FUNCTION_BLOCK FB_AdjustablePump IMPLEMENTS I_AdjustablePump

VAR
	bRunning : BOOL;
	fTotalVolume : REAL;
	fFlowRate : REAL := 20;
END_VAR

IF bRunning THEN
	fTotalVolume := fTotalVolume + fFlowRate;
END_IF

{warning 'add method implementation '}
METHOD GetFlowRate : REAL
GetFlowRate := fFlowRate;
END_METHOD

{warning 'add method implementation '}
METHOD GetTotalVolume : REAL
GetTotalVolume := fTotalVolume;
END_METHOD

METHOD SetFlowRate : BOOL
VAR_INPUT
	fNewRate : REAL;
END_VAR
fFlowRate := fNewRate;
END_METHOD

{warning 'add method implementation '}
METHOD Start : BOOL
Start := bRunning := TRUE;
END_METHOD

{warning 'add method implementation '}
METHOD Stop : BOOL
bRunning := FALSE;
END_METHOD

END_FUNCTION_BLOCK

(* stored: Version 1.1.0.1, ProductVersion 3.1.4024.16
   POU FB_AdjustablePump: Id {47ee60e1-54f9-4251-a115-40bdc03eaf9f}, SpecialFunc None
   Method GetFlowRate: Id {9081578a-d6ae-49d4-94f2-f41e166fc8dd}
   Method GetTotalVolume: Id {e8f654c5-f976-4a0b-a3bb-4e16d44c6672}
   Method SetFlowRate: Id {faee0fa6-0dbe-45b4-9bcc-c2da348c8215}
   Method Start: Id {ee90187c-98f6-49e2-96ab-50df4b18cc2d}
   Method Stop: Id {0d41d133-f600-4634-8863-771694af5da7} *)
